# EPICS autosave request: iocBoot/sioc-bc2b-bl01/blen_manual.req
file "manual.req" AREA=BC2B,POS=950,INST=BZ21BA
file "manual.req" AREA=BC2B,POS=950,INST=BZ21BB
